PROGRAM MAIN
VAR
END_VAR

END_PROGRAM

(* stored: Version 1.1.0.1
   POU MAIN: Id {29181515-19d8-4b8d-bbbf-5a8a6c9d7738} *)
